TYPE HMI_PROVIDER_HW_IO :
STRUCT
	stIn	: HMI_PROVIDER_HW_IN;
	stOut	: HMI_PROVIDER_HW_OUT;
END_STRUCT
END_TYPE

(* stored: Version 1.1.0.1, ProductVersion 3.1.4024.12
   DUT HMI_PROVIDER_HW_IO: Id {6f31cdcd-4e42-42c4-8af9-629c69b20c4b} *)
